Staubli VAL3: GetWeldReturn.pgx

public program GetWeldReturn(point& x_pCut[], point& x_pMC[], bool& x_bMC[], num x_nId, num& x_nReturnId, num x_nLength, bool& x_bRes)
  local num l_nNum
  local trsf l_trBuff[3]
  local trsf l_trTe
  local num l_nArc
  local num l_nLength
  local num l_nWeld
begin
  //获得回退点的MOVEID



  x_bRes=false
  x_nReturnId=-1
  if size(x_pCut)!=size(x_pMC) or size(x_pCut)!=size(x_bMC) or size(x_bMC)<(x_nId-1) or x_nLength<=0
    return
  endIf

  //如果只有一个点，则退出
   if size(x_bMC)==1
    x_bRes=true
    return
  endIf

  if roundDown(x_nId)==roundUp(x_nId)
      x_nId=x_nId+0.00001
  endIf


  //多于一个点进行计算
  l_nLength=0
  for l_nNum=1 to roundDown(x_nId)


    if !x_bMC[l_nNum]
      l_nArc=distance(x_pCut[l_nNum-1].trsf,x_pCut[l_nNum].trsf)

    else
      l_trBuff[0]=x_pCut[l_nNum-1].trsf
      l_trBuff[1]=x_pMC[l_nNum].trsf
      l_trBuff[2]=x_pCut[l_nNum].trsf
      //获取圆弧长度
      call GetArcLength(l_trBuff,l_nArc,x_bRes)
      if !x_bRes
        return
      endIf
    endIf

    //取余
    if l_nNum==roundDown(x_nId)
      l_nLength=(x_nId-l_nNum)*l_nArc+l_nLength
    else
      l_nLength=l_nLength+l_nArc
    endIf
  endFor

 // popUpMsg(toString(".3",l_nLength))
  //需要达到点的号码
  if l_nLength<=x_nLength
    x_nReturnId=1
      x_bRes=true
    return
  else
    l_nWeld=l_nLength-x_nLength
  endIf



  l_nLength=0
  for l_nNum=1 to roundUp(x_nId)


    if !x_bMC[l_nNum]
      l_nArc=distance(x_pCut[l_nNum-1].trsf,x_pCut[l_nNum].trsf)

    else
      l_trBuff[0]=x_pCut[l_nNum-1].trsf
      l_trBuff[1]=x_pMC[l_nNum].trsf
      l_trBuff[2]=x_pCut[l_nNum].trsf
      //获取圆弧长度
      call GetArcLength(l_trBuff,l_nArc,x_bRes)
      if !x_bRes
        return
      endIf
    endIf



    if l_nNum==roundUp(x_nId)-1
      l_nLength=(x_nId-roundDown(x_nId))*l_nArc+l_nLength
    else
      l_nLength=l_nLength+l_nArc
    endIf

    if l_nLength>=l_nWeld
      x_nReturnId=l_nNum-1-(l_nLength-l_nWeld)/l_nArc

        x_bRes=true
      return
    endIf
  endFor

  x_bRes=false

end
